(* Logix 5000 project; controller TEC_81 vendor 1 type 14 code 148 rev 36.11; software revision 36.00; part 3 of 4 *)
(* tags used below, declared in another part *)
   AbrirInterlock_conveyor_Safety : BOOL;   // Mapped green button for interlock 2 opening
   AbrirInterlock_Principal_Safety : BOOL;   // Mapped green button for interlock 1 opening
   Axis_1 : AXIS_CIP_DRIVE;
   Axis_2 : AXIS_CIP_DRIVE;   // Almacen 2
   Cmd_Axis_2 : BOOL;
   Cmd_Robot_Conv_1 : BOOL;
   Cmd_Robot_Conv_2 : BOOL;
   Cmd_YPickSafe_Alm1 : BOOL;
   Cmd_YPlaceSafe_Alm1 : BOOL;
   Cmd_YSafePos_Alm1 : BOOL;
   Cmd_YtoYOff_Alm1 : BOOL;
   Cmd_YtoYPick_Alm1 : BOOL;
   Cmd_YtoYPlace_Alm1 : BOOL;
   Cmd_YtoYPlaceOffset_Alm1 : BOOL;
   Consumeded_Signals_Conveyor_1_TEC_81 : DINT;
   Conveyor_1_Tomar_Pieza : BOOL;   // Señal del Conveyor 1 para Tomar Pieza Iniciar Ciclo
   Conveyor_2_Tomar_Pieza : BOOL;   // Señal del Conveyor 2 para Tomar Pieza Iniciar Ciclo
   EStops_OK : BOOL;   // E-Stop Close Loop Indicator
   EStops_OK_External : DINT;
   From_Robot : FromRobot_v02;
   From_Wh2 : DINT;
   FromStorage1 : DINT;
   Home_Sensor : BOOL;
   Input_Reset_Almacen_1 : BOOL;
   Input_Reset_almacen_2 : BOOL;
   Input_Reset_Principal : BOOL;
   Input_Reset_Salida_1 : BOOL;
   Interlocks_Ok : BOOL;   // Interlocks Close Loop Indicator
   LigthCurtain_ok : BOOL;   // Light Curtains Close Loop Indicator
   MC_1_EStop : DCI_STOP;   // Status of E-Stop 1
   MC_1_EStop_Status : BOOL;   // General status of inputs
   MC_1_Interlock : DCI_STOP;   // Status of Interlock 1
   MC_1_Interlock_Status : BOOL;   // General status of inputs
   MC_1_LigthCurtain : DCI_STOP;   // Status of Light Curtain 1
   MC_1_LigthCurtain_Status : BOOL;   // General status of inputs
   MC_2_EStop : DCI_STOP;   // Status of E-Stop 2
   MC_2_EStop_Status : BOOL;   // General status of inputs
   MC_2_Interlock : DCI_STOP;   // Status of Interlock 2
   MC_2_Interlock_Status : BOOL;   // General status of inputs
   MC_2_LightCurtain_Status : BOOL;   // General status of inputs
   MC_2_LigthCurtain : DCI_STOP;   // Status of Light Curtain 2
   MC_3_EStop : DCI_STOP;   // Status of E-Stop 3
   MC_3_EStop_Status : BOOL;   // General status of inputs
   MC_4_EStop : DCI_STOP;   // Status of E-Stop 4
   MC_4_EStop_Status : BOOL;   // General status of inputs
   MC_5_EStop : DCI_STOP;   // Status of E-Stop 5
   MC_5_EStop_Status : BOOL;   // General status of inputs
   ok : BOOL;
   Ons : INT;
   Operation_Mode : BOOL;   // Operation Mode for HMI
   Produced_Signals_TEC_81_Conveyor_1 : DINT;
   Reset_Almacen_1 : BOOL;
   Reset_almacen_2 : BOOL;
   Reset_Principal : BOOL;
   Reset_Salida_1 : BOOL;
   Retorno_Pieza_A_Conveyor_1 : BOOL;
   Robot_Step : DINT;
   Safety_FromTEC81 : Safety;
   Signal_Fanuc_Tomar_Pieza_Conv_1 : BOOL;   // Señal para Tomar pieza desde el Conveyor 1 Hacia CNC
   Storage_1_Y_ActualPosition : REAL;
   Storage_2_Y_ActualPosition : REAL;
   Tec81_to_Wh2 : DINT;
   test_com : BOOL;   // bit e comunicacion
   TEst_Leaa_Sfty : DINT;
   TT : BOOL;
(* MainProgram, continued *)

ROUTINE _08_Outputs   (* ladder *)
END_ROUTINE

ROUTINE _09_Resets   (* ladder *)
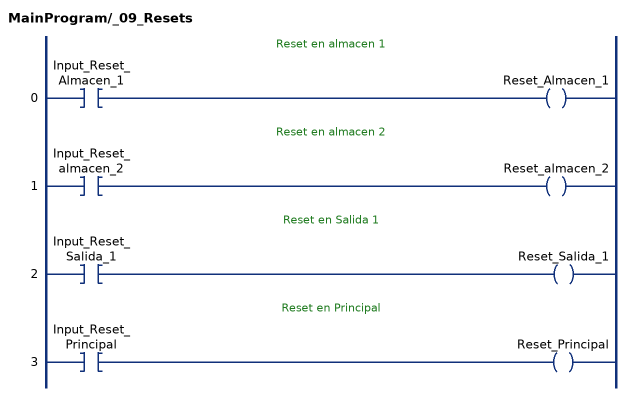
   // Reset en almacen 1
   0: XIC(Input_Reset_Almacen_1)OTE(Reset_Almacen_1);
   // Reset en almacen 2
   1: XIC(Input_Reset_almacen_2)OTE(Reset_almacen_2);
   // Reset en Salida 1
   2: XIC(Input_Reset_Salida_1)OTE(Reset_Salida_1);
   // Reset en Principal
   3: XIC(Input_Reset_Principal)OTE(Reset_Principal);
END_ROUTINE

ROUTINE _10_ExternalComm   (* ladder *)
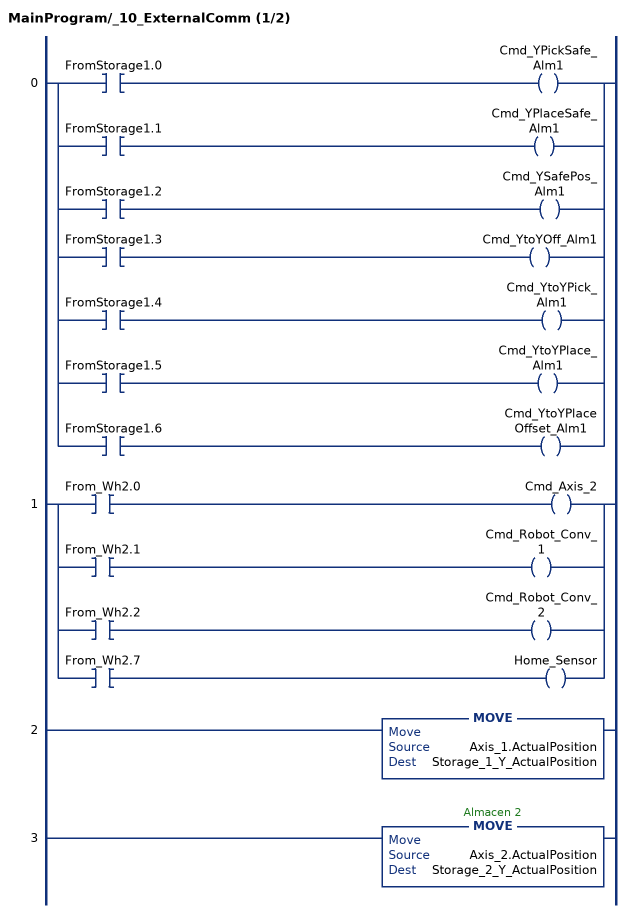
   0: [XIC(FromStorage1.0) OTE(Cmd_YPickSafe_Alm1) ,XIC(FromStorage1.1) OTE(Cmd_YPlaceSafe_Alm1) ,XIC(FromStorage1.2) OTE(Cmd_YSafePos_Alm1) ,XIC(FromStorage1.3) OTE(Cmd_YtoYOff_Alm1) ,XIC(FromStorage1.4) OTE(Cmd_YtoYPick_Alm1) ,XIC(FromStorage1.5) OTE(Cmd_YtoYPlace_Alm1) ,XIC(FromStorage1.6) OTE(Cmd_YtoYPlaceOffset_Alm1) ];
   1: [XIC(From_Wh2.0) OTE(Cmd_Axis_2) ,XIC(From_Wh2.1) OTE(Cmd_Robot_Conv_1) ,XIC(From_Wh2.2) OTE(Cmd_Robot_Conv_2) ,XIC(From_Wh2.7) OTE(Home_Sensor) ];
   2: MOVE(Axis_1.ActualPosition,Storage_1_Y_ActualPosition);
   3: MOVE(Axis_2.ActualPosition,Storage_2_Y_ActualPosition);
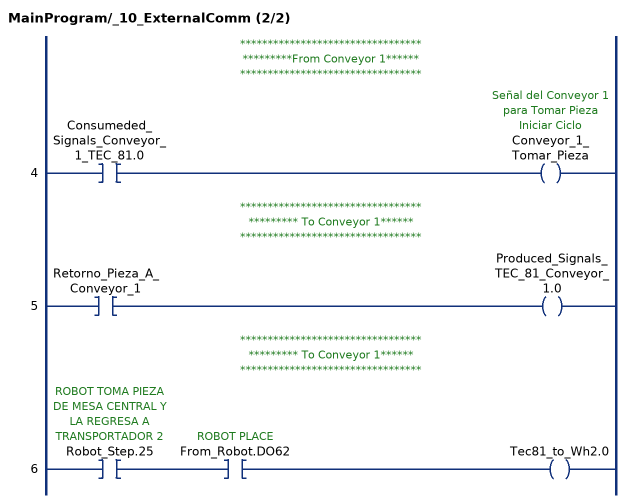
   // *********************************
   // *********From Conveyor 1******
   // *********************************
   4: XIC(Consumeded_Signals_Conveyor_1_TEC_81.0)OTE(Conveyor_1_Tomar_Pieza);
   // *********************************
   // ********* To Conveyor 1******
   // *********************************
   5: XIC(Retorno_Pieza_A_Conveyor_1)OTE(Produced_Signals_TEC_81_Conveyor_1.0);
   // *********************************
   // ********* To Conveyor 1******
   // *********************************
   6: XIC(Robot_Step.25)XIC(From_Robot.DO62)OTE(Tec81_to_Wh2.0);
END_ROUTINE

ROUTINE _11_External   (* ladder *)
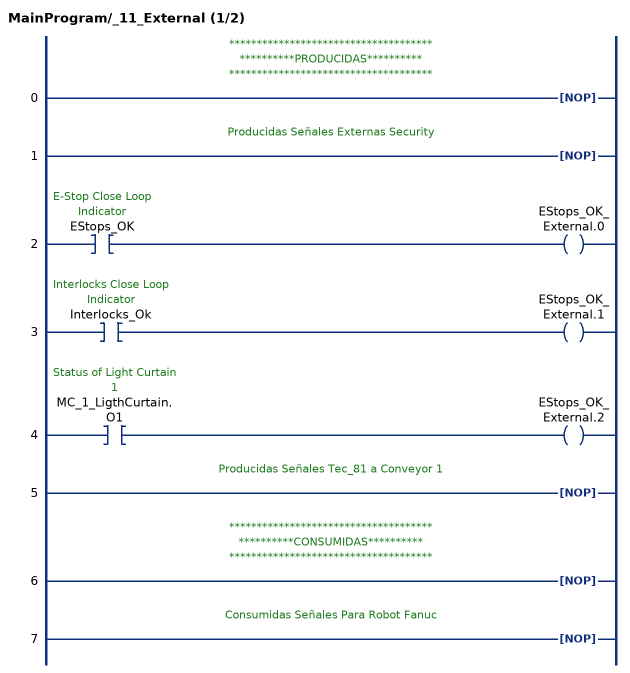
   // *************************************
   // **********PRODUCIDAS**********
   // *************************************
   0: NOP();
   // Producidas Señales Externas Security
   1: NOP();
   2: XIC(EStops_OK)OTE(EStops_OK_External.0);
   3: XIC(Interlocks_Ok)OTE(EStops_OK_External.1);
   4: XIC(MC_1_LigthCurtain.O1)OTE(EStops_OK_External.2);
   // Producidas Señales Tec_81 a Conveyor 1
   5: NOP();
   // *************************************
   // **********CONSUMIDAS**********
   // *************************************
   6: NOP();
   // Consumidas Señales Para Robot Fanuc
   7: NOP();
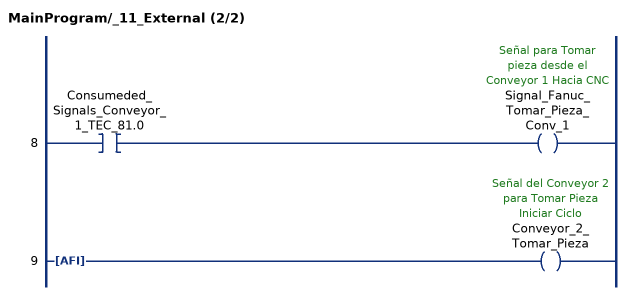
   8: XIC(Consumeded_Signals_Conveyor_1_TEC_81.0)OTE(Signal_Fanuc_Tomar_Pieza_Conv_1);
   9: AFI()OTE(Conveyor_2_Tomar_Pieza);
END_ROUTINE

ROUTINE MainRoutine   (* ladder *)
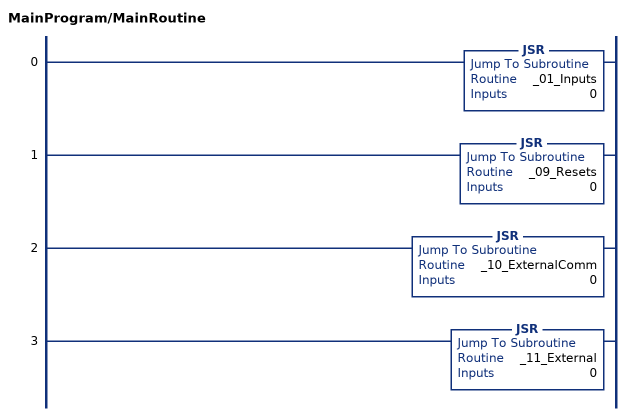
   0: JSR(_01_Inputs,0);
   1: JSR(_09_Resets,0);
   2: JSR(_10_ExternalComm,0);
   3: JSR(_11_External,0);
END_ROUTINE
END_PROGRAM

PROGRAM SafetyProgram   (* main routine MainRoutine, safety *)
VAR
   dummy : BOOL;
   Lasers_OK : BOOL;   // Laser Scanner Close Loop Indicator
   LS_1 : DCI_STOP;   // Status of Laser Scanner 1
   LS_1_Status : BOOL := 1;   // General status of inputs
   LS_2 : DCI_STOP;   // Status of Laser Scanner 2
   LS_2_Status : BOOL := 1;   // General status of inputs
   Mat_1 : DCI_STOP;   // Status of Safety Mat 1
   Mat_1_Status : BOOL := 1;   // General status of inputs
   ONS_Laser_1 : BOOL;   // One time execution for reset
   ONS_Laser_2 : BOOL;   // One time execution for reset
   ONS_Mat_1 : BOOL;   // One time execution for reset
   Output_Enable_Laser_1 : BOOL;   // General status of Laser 1
   Output_Enable_Laser_2 : BOOL;   // General status of Laser 2
   Output_Enable_Mat_1 : BOOL;   // General status of Mat 1
   Safety_Close_Loop_ok : BOOL;   // General Safety Indicator
   Safety_Latch_Timer : TIMER;
   Safety_Mat_ok : BOOL;   // Safety Mat Close Loop Indicator
   Safety_Reset_General : BOOL;   // Unified General Reset
   test_1 : BOOL;
   test_21 : BOOL;
   TOF_STO_KinetixStorage1 : TIMER;
END_VAR

ROUTINE Estops   (* ladder *)
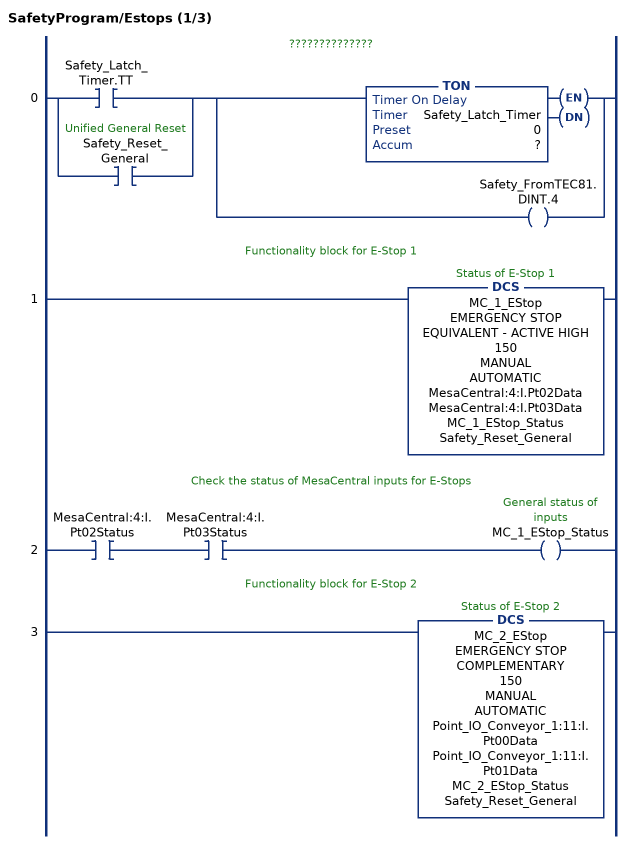
   // ??????????????
   0: [XIC(Safety_Latch_Timer.TT) ,XIC(Safety_Reset_General) ][TON(Safety_Latch_Timer,?,?) ,OTE(Safety_FromTEC81.DINT.4) ];
   // Functionality block for E-Stop 1
   1: DCS(MC_1_EStop,EMERGENCY STOP,EQUIVALENT - ACTIVE HIGH,150,MANUAL,AUTOMATIC,MesaCentral:4:I.Pt02Data,MesaCentral:4:I.Pt03Data,MC_1_EStop_Status,Safety_Reset_General);
   // Check the status of MesaCentral inputs for E-Stops
   2: XIC(MesaCentral:4:I.Pt02Status)XIC(MesaCentral:4:I.Pt03Status)OTE(MC_1_EStop_Status);
   // Functionality block for E-Stop 2
   3: DCS(MC_2_EStop,EMERGENCY STOP,COMPLEMENTARY,150,MANUAL,AUTOMATIC,Point_IO_Conveyor_1:11:I.Pt00Data,Point_IO_Conveyor_1:11:I.Pt01Data,MC_2_EStop_Status,Safety_Reset_General);
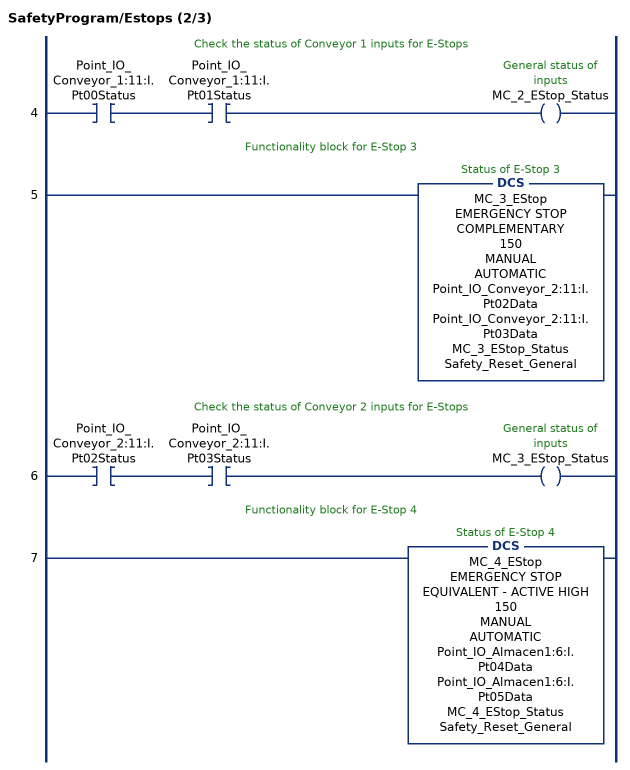
   // Check the status of Conveyor 1 inputs for E-Stops
   4: XIC(Point_IO_Conveyor_1:11:I.Pt00Status)XIC(Point_IO_Conveyor_1:11:I.Pt01Status)OTE(MC_2_EStop_Status);
   // Functionality block for E-Stop 3
   5: DCS(MC_3_EStop,EMERGENCY STOP,COMPLEMENTARY,150,MANUAL,AUTOMATIC,Point_IO_Conveyor_2:11:I.Pt02Data,Point_IO_Conveyor_2:11:I.Pt03Data,MC_3_EStop_Status,Safety_Reset_General);
   // Check the status of Conveyor 2 inputs for E-Stops
   6: XIC(Point_IO_Conveyor_2:11:I.Pt02Status)XIC(Point_IO_Conveyor_2:11:I.Pt03Status)OTE(MC_3_EStop_Status);
   // Functionality block for E-Stop 4
   7: DCS(MC_4_EStop,EMERGENCY STOP,EQUIVALENT - ACTIVE HIGH,150,MANUAL,AUTOMATIC,Point_IO_Almacen1:6:I.Pt04Data,Point_IO_Almacen1:6:I.Pt05Data,MC_4_EStop_Status,Safety_Reset_General);
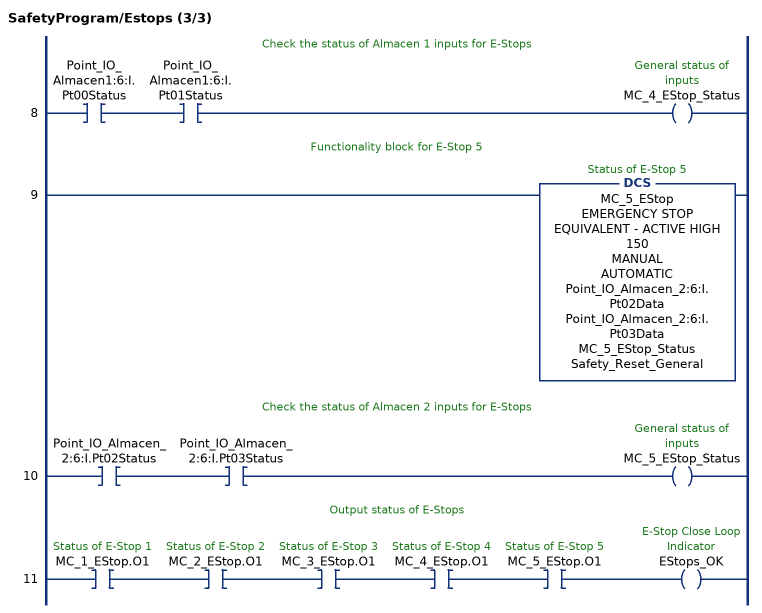
   // Check the status of Almacen 1 inputs for E-Stops
   8: XIC(Point_IO_Almacen1:6:I.Pt00Status)XIC(Point_IO_Almacen1:6:I.Pt01Status)OTE(MC_4_EStop_Status);
   // Functionality block for E-Stop 5
   9: DCS(MC_5_EStop,EMERGENCY STOP,EQUIVALENT - ACTIVE HIGH,150,MANUAL,AUTOMATIC,Point_IO_Almacen_2:6:I.Pt02Data,Point_IO_Almacen_2:6:I.Pt03Data,MC_5_EStop_Status,Safety_Reset_General);
   // Check the status of Almacen 2 inputs for E-Stops
   10: XIC(Point_IO_Almacen_2:6:I.Pt02Status)XIC(Point_IO_Almacen_2:6:I.Pt03Status)OTE(MC_5_EStop_Status);
   // Output status of E-Stops
   11: XIC(MC_1_EStop.O1)XIC(MC_2_EStop.O1)XIC(MC_3_EStop.O1)XIC(MC_4_EStop.O1)XIC(MC_5_EStop.O1)OTE(EStops_OK);
END_ROUTINE

ROUTINE External_COMM   (* ladder *)
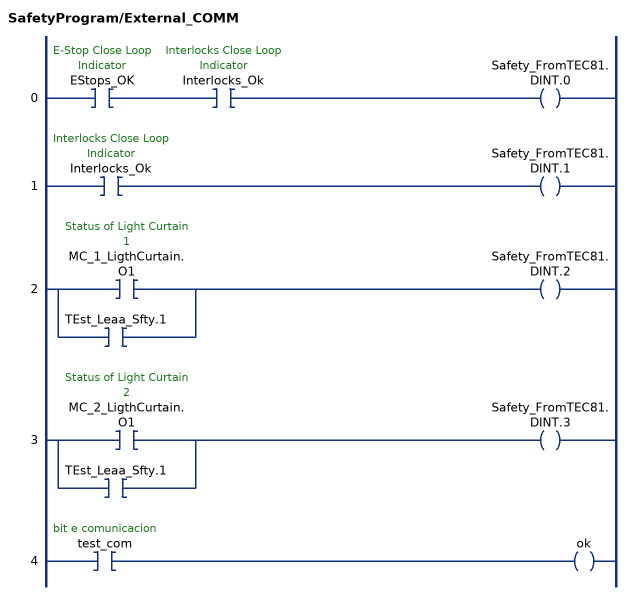
   0: XIC(EStops_OK)XIC(Interlocks_Ok)OTE(Safety_FromTEC81.DINT.0);
   1: XIC(Interlocks_Ok)OTE(Safety_FromTEC81.DINT.1);
   2: [XIC(MC_1_LigthCurtain.O1) ,XIC(TEst_Leaa_Sfty.1) ]OTE(Safety_FromTEC81.DINT.2);
   3: [XIC(MC_2_LigthCurtain.O1) ,XIC(TEst_Leaa_Sfty.1) ]OTE(Safety_FromTEC81.DINT.3);
   4: XIC(test_com)OTE(ok);
END_ROUTINE

ROUTINE Fanuc   (* ladder *)
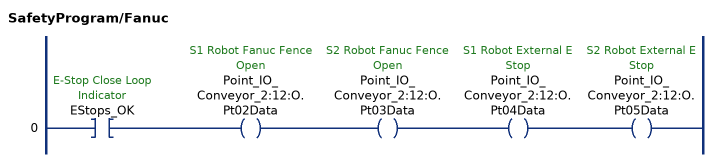
   0: XIC(EStops_OK)OTE(Point_IO_Conveyor_2:12:O.Pt02Data)OTE(Point_IO_Conveyor_2:12:O.Pt03Data)OTE(Point_IO_Conveyor_2:12:O.Pt04Data)OTE(Point_IO_Conveyor_2:12:O.Pt05Data);
END_ROUTINE

ROUTINE Interlocks   (* ladder *)
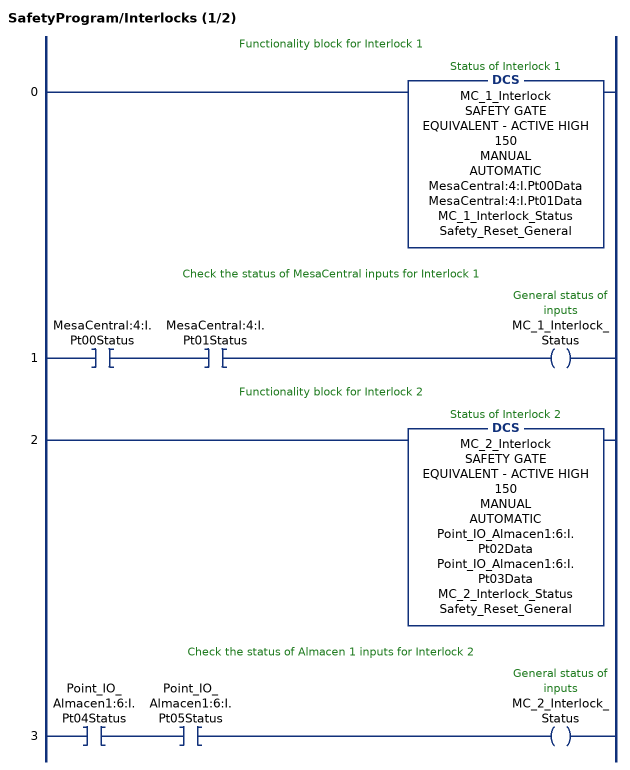
   // Functionality block for Interlock 1
   0: DCS(MC_1_Interlock,SAFETY GATE,EQUIVALENT - ACTIVE HIGH,150,MANUAL,AUTOMATIC,MesaCentral:4:I.Pt00Data,MesaCentral:4:I.Pt01Data,MC_1_Interlock_Status,Safety_Reset_General);
   // Check the status of MesaCentral inputs for Interlock 1
   1: XIC(MesaCentral:4:I.Pt00Status)XIC(MesaCentral:4:I.Pt01Status)OTE(MC_1_Interlock_Status);
   // Functionality block for Interlock 2
   2: DCS(MC_2_Interlock,SAFETY GATE,EQUIVALENT - ACTIVE HIGH,150,MANUAL,AUTOMATIC,Point_IO_Almacen1:6:I.Pt02Data,Point_IO_Almacen1:6:I.Pt03Data,MC_2_Interlock_Status,Safety_Reset_General);
   // Check the status of Almacen 1 inputs for Interlock 2
   3: XIC(Point_IO_Almacen1:6:I.Pt04Status)XIC(Point_IO_Almacen1:6:I.Pt05Status)OTE(MC_2_Interlock_Status);
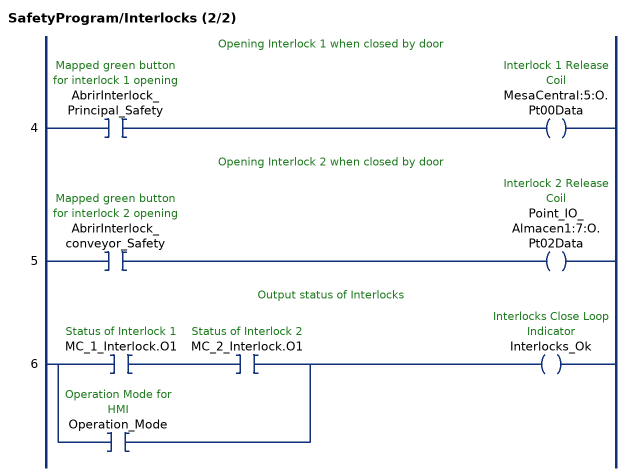
   // Opening Interlock 1 when closed by door
   4: XIC(AbrirInterlock_Principal_Safety)OTE(MesaCentral:5:O.Pt00Data);
   // Opening Interlock 2 when closed by door
   5: XIC(AbrirInterlock_conveyor_Safety)OTE(Point_IO_Almacen1:7:O.Pt02Data);
   // Output status of Interlocks
   6: [XIC(MC_1_Interlock.O1) XIC(MC_2_Interlock.O1) ,XIC(Operation_Mode) ]OTE(Interlocks_Ok);
END_ROUTINE

ROUTINE Laser_Scanner   (* ladder *)
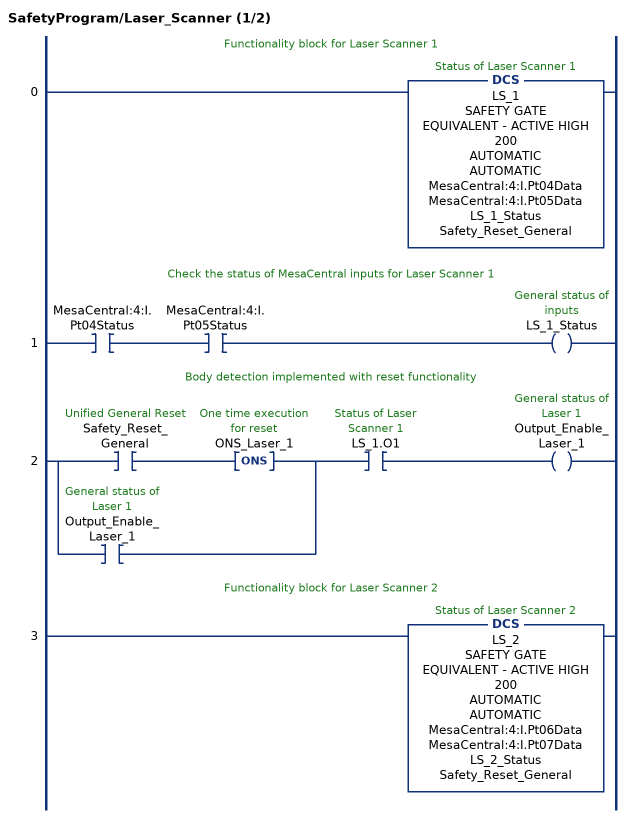
   // Functionality block for Laser Scanner 1
   0: DCS(LS_1,SAFETY GATE,EQUIVALENT - ACTIVE HIGH,200,AUTOMATIC,AUTOMATIC,MesaCentral:4:I.Pt04Data,MesaCentral:4:I.Pt05Data,LS_1_Status,Safety_Reset_General);
   // Check the status of MesaCentral inputs for Laser Scanner 1
   1: XIC(MesaCentral:4:I.Pt04Status)XIC(MesaCentral:4:I.Pt05Status)OTE(LS_1_Status);
   // Body detection implemented with reset functionality
   2: [XIC(Safety_Reset_General) ONS(ONS_Laser_1) ,XIC(Output_Enable_Laser_1) ]XIC(LS_1.O1)OTE(Output_Enable_Laser_1);
   // Functionality block for Laser Scanner 2
   3: DCS(LS_2,SAFETY GATE,EQUIVALENT - ACTIVE HIGH,200,AUTOMATIC,AUTOMATIC,MesaCentral:4:I.Pt06Data,MesaCentral:4:I.Pt07Data,LS_2_Status,Safety_Reset_General);
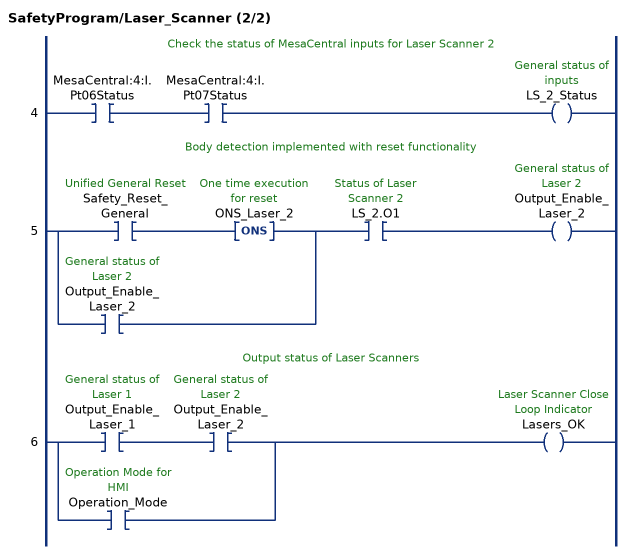
   // Check the status of MesaCentral inputs for Laser Scanner 2
   4: XIC(MesaCentral:4:I.Pt06Status)XIC(MesaCentral:4:I.Pt07Status)OTE(LS_2_Status);
   // Body detection implemented with reset functionality
   5: [XIC(Safety_Reset_General) ONS(ONS_Laser_2) ,XIC(Output_Enable_Laser_2) ]XIC(LS_2.O1)OTE(Output_Enable_Laser_2);
   // Output status of Laser Scanners
   6: [XIC(Output_Enable_Laser_1) XIC(Output_Enable_Laser_2) ,XIC(Operation_Mode) ]OTE(Lasers_OK);
END_ROUTINE

ROUTINE LigthCurrtains   (* ladder *)
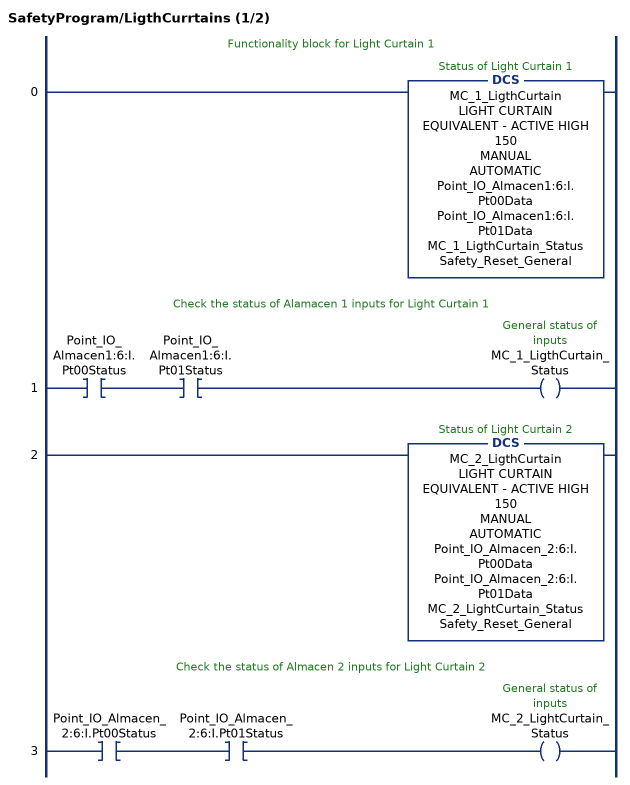
   // Functionality block for Light Curtain 1
   0: DCS(MC_1_LigthCurtain,LIGHT CURTAIN,EQUIVALENT - ACTIVE HIGH,150,MANUAL,AUTOMATIC,Point_IO_Almacen1:6:I.Pt00Data,Point_IO_Almacen1:6:I.Pt01Data,MC_1_LigthCurtain_Status,Safety_Reset_General);
   // Check the status of Alamacen 1 inputs for Light Curtain 1
   1: XIC(Point_IO_Almacen1:6:I.Pt00Status)XIC(Point_IO_Almacen1:6:I.Pt01Status)OTE(MC_1_LigthCurtain_Status);
   2: DCS(MC_2_LigthCurtain,LIGHT CURTAIN,EQUIVALENT - ACTIVE HIGH,150,MANUAL,AUTOMATIC,Point_IO_Almacen_2:6:I.Pt00Data,Point_IO_Almacen_2:6:I.Pt01Data,MC_2_LightCurtain_Status,Safety_Reset_General);
   // Check the status of Almacen 2 inputs for Light Curtain 2
   3: XIC(Point_IO_Almacen_2:6:I.Pt00Status)XIC(Point_IO_Almacen_2:6:I.Pt01Status)OTE(MC_2_LightCurtain_Status);
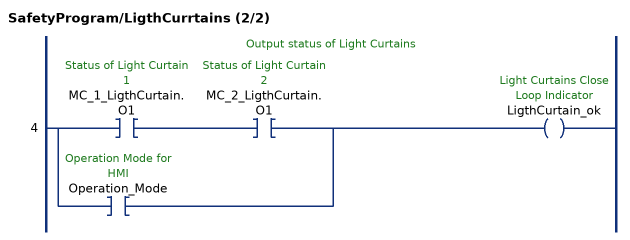
   // Output status of Light Curtains
   4: [XIC(MC_1_LigthCurtain.O1) XIC(MC_2_LigthCurtain.O1) ,XIC(Operation_Mode) ]OTE(LigthCurtain_ok);
END_ROUTINE

ROUTINE MainRoutine   (* ladder *)
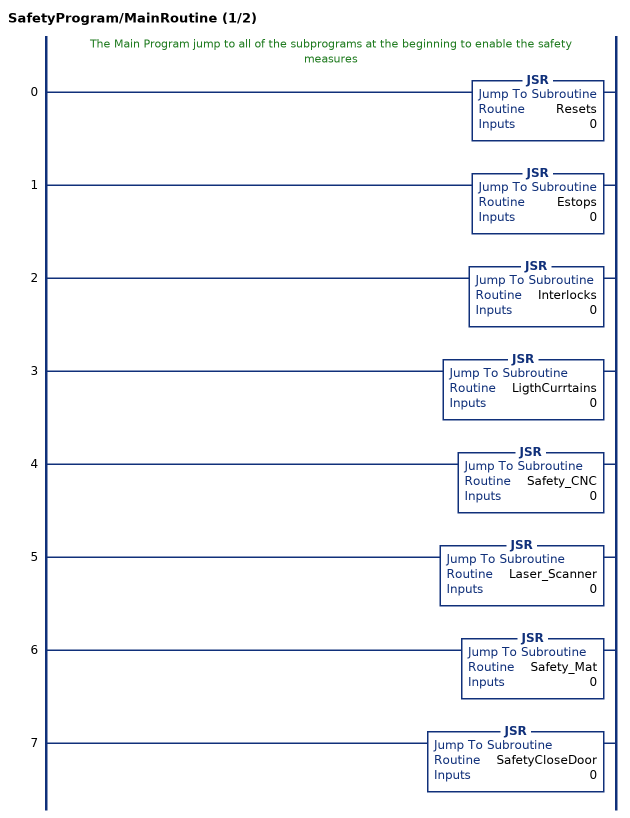
   // The Main Program jump to all of the subprograms at the beginning to enable the safety measures
   0: JSR(Resets,0);
   1: JSR(Estops,0);
   2: JSR(Interlocks,0);
   3: JSR(LigthCurrtains,0);
   4: JSR(Safety_CNC,0);
   5: JSR(Laser_Scanner,0);
   6: JSR(Safety_Mat,0);
   7: JSR(SafetyCloseDoor,0);
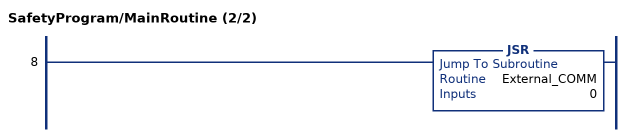
   8: JSR(External_COMM,0);
END_ROUTINE
